# EPICS substitutions: modules/event/evrSupport/Db/ioc/IOC-LR20-LS01evr.substitutions
#==============================================================================
#
# Abs:  LCLS EVR IOC records for LR20 LS01
#
# Name: IOC-LR20-LS01evr.substitutions
#
#==============================================================================
#
file evrLSXX.db
{
pattern { DEVICE        }
	{ EVR:LR20:LS01 }
}
